FUNCTION_BLOCK BTN_LGHT (* Composite Function Block Type *)
  (* Standard: 61499-2 *)
  (* Version 0.2, 2003-12-05, JHC, Rockwell Automation, Renamed from NEWCOMPFB. *)
  (* Version 0.1, 2002-01-08, JHC, Rockwell Automation, Added DLY FB as example. *)
  (* Version 0.0, 2000-05-27, JHC, Rockwell Automation *)
  (* Compiler header: package fb.rt.vhmi;import fb.rt.hmi.*; *)
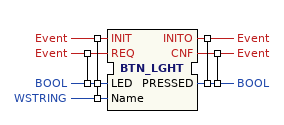
  EVENT_INPUT
    INIT WITH LED, Name; (* Initialization Request *)
    REQ WITH LED; (* Normal Execution Request *)
  END_EVENT
  EVENT_OUTPUT
    INITO WITH PRESSED; (* Initialization Confirm *)
    CNF WITH PRESSED; (* Execution Confirmation *)
  END_EVENT
  VAR_INPUT
    LED : BOOL; (* Input event qualifier *)
    Name : WSTRING;
  END_VAR
  VAR_OUTPUT
    PRESSED : BOOL; (* Output event qualifier *)
  END_VAR
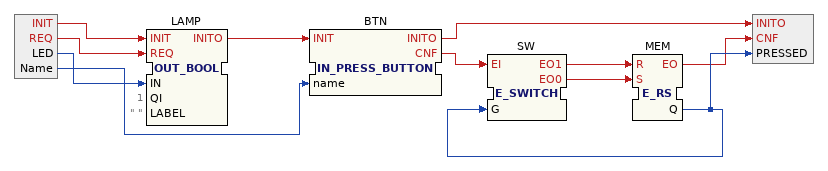
  FBS
    LAMP : OUT_BOOL(QI := 1, LABEL := " ");
    MEM : E_RS;
    BTN : IN_PRESS_BUTTON;
    SW : E_SWITCH;
  END_FBS
  EVENT_CONNECTIONS
    BTN.INITO TO INITO;
    LAMP.INITO TO BTN.INIT;
    INIT TO LAMP.INIT;
    REQ TO LAMP.REQ;
    MEM.EO TO CNF;
    SW.EO1 TO MEM.R;
    SW.EO0 TO MEM.S;
    BTN.CNF TO SW.EI;
  END_CONNECTIONS
  DATA_CONNECTIONS
    Name TO BTN.name;
    MEM.Q TO PRESSED;
    LED TO LAMP.IN;
    MEM.Q TO SW.G;
  END_CONNECTIONS
END_FUNCTION_BLOCK
